// 编辑数据表的字段和类型



  TYPE ST_ProdEntry :


STRUCT
 ID :


UDINT;


JS :


string(50);


FTPDOWN :


BOOL;


DATAEXPORT :


BOOL;


DICTEDIT :


BOOL;


CREATETAB :


BOOL;


END_STRUCT


END_TYPE

(* stored: Version 1.1.0.1, ProductVersion 3.1.4024.16
   DUT ST_ProdEntry: Id {b5ef3a82-e286-4b34-be9a-84be3468753a} *)
